// TIA Portal V21 export
// export: Created 2026-07-28T16:54:16.2255313Z, ExportSetting WithDefaults, DisplayName Totally Integrated Automation Portal, DisplayVersion V21, DisplayName SINAMICS Startdrive Advanced, DisplayVersion V21, DisplayName SINAMICS Startdrive G110M, G120, G120C, G120D, G120P, G115D, DisplayVersion V21, DisplayName SINAMICS Startdrive G130, G150, S120, S150, G200, G220, S200, S210, S220, Innomotics MVD, DisplayVersion V21, DisplayName STEP 7 Professional, DisplayVersion V21, DisplayName STEP 7 Safety, DisplayVersion V21, DisplayName Tech WebApplication, DisplayVersion V21, DisplayName WinCC Basic/Comfort/Advanced, DisplayVersion V21, DisplayName WinCC Professional, DisplayVersion V21, DisplayName WinCC Unified, DisplayVersion V21
TYPE "ValvDados"
// stored: IsFailsafeCompliant false
   STRUCT
      STS_VALVULA_ABERTA : Bool;   // fim de curso aberto
      STS_VALVULA_FECHADA : Bool;   // fim de curso fechado
      STS_MODO_LOCAL : Bool;   // chave do atuador em local
      STS_MODO_REMOTO : Bool;   // chave do atuador em remoto
      STS_VALVULA_AUTOMATICO : Bool;   // remoto + habilitada pelo processo
      STS_FALHA_TORQUE_ABERTURA : Bool;
      STS_FALHA_TORQUE_FECHAMENTO : Bool;
      STS_FALHA_TEMPO_CURSO : Bool;   // nao chegou ao fim de curso no tempo
      STS_VALVULA_FEEDBACK_POSICAO : Int;   // posicao 0..27648 (raw) em valvula proporcional --- comandos ---
      CMD_VALVULA_ABRE : Bool;
      CMD_VALVULA_FECHA : Bool;
      CMD_MANUAL : Bool;
      CMD_RESET_FALHA : Bool;
      SP_SETPOINT_MANUAL : Real;   // posicao desejada em manual [%]
      SP_SETPOINT_AUTO : Real;   // posicao desejada em automatico [%] --- parametros de cadastro ---
      SP_TEMPO_CURSO : Real;   // [s] tempo nominal de abertura/fechamento --- reserva ---
      RESERVA_BOOL_01 : Bool;
      RESERVA_BOOL_02 : Bool;
      RESERVA_INT_01 : Int;
      RESERVA_REAL_01 : Real;
   END_STRUCT;
END_TYPE
